{attribute addProperty BoxType "AX8620-0000-0029"}
{attribute addProperty Id "PSM_Controlword_for_axisAT %I*PSM_Controlword_for_axis_59B039C11620WcStateAT %I*WcState_98A4DF7520.250InfoDataAT %I*InfoData_0BDED7BF144180"}
{attribute addProperty CRC "4182654517"}
{attribute addProperty SizeInBites "162"}
{attribute addProperty SizeInBytes "20.25"}
TYPE AX8620_4A923142 :
STRUCT
	{attribute addProperty Name "PSM_Controlword_for_axis"}
	PSM_Controlword_for_axis : PSM_Controlword_for_axis_59B039C1;
	{attribute addProperty Name "WcState"}
	WcState : WcState_98A4DF75;
	{attribute addProperty Name "InfoData"}
	InfoData : InfoData_0BDED7BF;
END_STRUCT
END_TYPE

(* stored: Version 1.2.0.0, ProductVersion 3.1.4024.9
   DUT AX8620_4A923142: Id {ffb784ab-6286-475b-8393-806237ce4818} *)
